{attribute 'qualified_only'}
VAR_GLOBAL
    //Message : FB_TcMessage;
END_VAR

(* stored: Version 1.1.0.1, ProductVersion 3.1.4024.4
   GVL GlobalVariables: Id {286734ed-0e51-4e1c-a2a6-a40cdf8eaf62} *)
